{attribute 'no_explicit_call' := 'MySingleton is a CLASS and must be accessed using methods or properties'}
FUNCTION_BLOCK MessageLogger IMPLEMENTS I_MessageLogger
VAR_STAT 	// VAR_STAT makes sure all new instances use the same initialized vars
	messageLogger					: I_MessageLogger;				
	messageLoggerSingleton			: POINTER TO MessageLoggerSingleton;
END_VAR

METHOD FB_exit : BOOL
VAR_INPUT
	bInCopyCode : BOOL; // if TRUE, the exit method is called for exiting an instance that is copied afterwards (online change).
END_VAR
// Delete the dynamic instance at FB_exit 
IF messageLoggerSingleton <> 0	THEN
	messageLogger := 0;					// Clear interface
	__DELETE(messageLoggerSingleton);	// Delete the instance
	messageLoggerSingleton:=0;			// Clear the pointer
END_IF
END_METHOD

METHOD FB_init : BOOL
VAR_INPUT
	bInitRetains : BOOL; // if TRUE, the retain variables are initialized (warm start / cold start)
	bInCopyCode : BOOL;  // if TRUE, the instance afterwards gets moved into the copy code (online change)
END_VAR
// first instance? 
IF messageLoggerSingleton = 0	THEN
	messageLoggerSingleton := __NEW(messageLoggerSingleton);
	messageLogger := messageLoggerSingleton^;
END_IF
END_METHOD

METHOD LogMessage : STRING
VAR_INPUT
	message			: STRING;
END_VAR
IF messageLogger <> 0 THEN
	messageLogger.LogMessage(message);
END_IF
END_METHOD

{warning 'add property implementation'}
PROPERTY message : STRING
GET
message := messageLogger.message;
END_GET
END_PROPERTY

END_FUNCTION_BLOCK

(* stored: Version 1.1.0.1, ProductVersion 3.1.4024.12
   POU MessageLogger: Id {1efae137-7a3a-4e0c-866d-49c9343a6747}, SpecialFunc None
   Method FB_exit: Id {ac91d9c2-bf66-4068-a24f-70354b3b2745}
   Method FB_init: Id {c1b2c753-7477-4d5a-bd89-3e2870801467}
   Method LogMessage: Id {b5e04c8e-02d8-4dd7-b341-2fd50157c5d3}
   Property message: Id {67119e77-db8e-4837-8895-a3b79092479d}
   Get Get: Id {5dea044f-85b1-4124-953d-21e28e237d44} *)
